LIN {X 0,Y 101.376,Z 372.445,A -85,B 0,C 180,E1 -29319.712,E2 -29319.712} C_VEL
LIN {X 0,Y 101.668,Z 372.001,A -85,B 0,C 180,E1 -29323.941,E2 -29323.941} C_VEL
LIN {X 0,Y 92.966,Z 374.596,A -85,B 0,C 180,E1 -29326.884,E2 -29326.884} C_VEL
LIN {X 0,Y 84.662,Z 376.417,A -85,B 0,C 180,E1 -29330.435,E2 -29330.435} C_VEL
LIN {X 0,Y 76.767,Z 377.474,A -85,B 0,C 180,E1 -29334.739,E2 -29334.739} C_VEL
LIN {X 0,Y 69.451,Z 377.857,A -85,B 0,C 180,E1 -29339.99,E2 -29339.99} C_VEL
LIN {X 0,Y 62.844,Z 377.562,A -85,B 0,C 180,E1 -29346.41,E2 -29346.41} C_VEL
LIN {X 0,Y 57.18,Z 376.524,A -85,B 0,C 180,E1 -29354.218,E2 -29354.218} C_VEL
LIN {X 0,Y 51.191,Z 373.837,A -85,B 0,C 180,E1 -29367.967,E2 -29367.967} C_VEL
LIN {X 0,Y 48.505,Z 369.652,A -85,B 0,C 180,E1 -29383.582,E2 -29383.582} C_VEL
LIN {X 0,Y 49.289,Z 364.241,A -85,B 0,C 180,E1 -29398.79,E2 -29398.79} C_VEL
LIN {X 0,Y 52.121,Z 358.398,A -85,B 0,C 180,E1 -29410.672,E2 -29410.672} C_VEL
LIN {X 0,Y 56.794,Z 350.599,A -85,B 0,C 180,E1 -29421.784,E2 -29421.784} C_VEL
LIN {X 0,Y 62.197,Z 342.135,A -85,B 0,C 180,E1 -29430.004,E2 -29430.004} C_VEL
LIN {X 0,Y 68.349,Z 332.145,A -85,B 0,C 180,E1 -29436.646,E2 -29436.646} C_VEL
LIN {X 0,Y 70.549,Z 328.315,A -85,B 0,C 180,E1 -29438.597,E2 -29438.597} C_VEL
LIN {X 0,Y 71.058,Z 326.204,A -85,B 0,C 180,E1 -29439.97,E2 -29439.97} C_VEL
LIN {X 0,Y 70.945,Z 321.655,A -85,B 0,C 180,E1 -29443.65,E2 -29443.65} C_VEL
LIN {X 0,Y 69.588,Z 315.642,A -85,B 0,C 180,E1 -29449.36,E2 -29449.36} C_VEL
LIN {X 0,Y 68.088,Z 310.944,A -85,B 0,C 180,E1 -29454.389,E2 -29454.389} C_VEL
LIN {X 0,Y 65.675,Z 304.781,A -85,B 0,C 180,E1 -29462.352,E2 -29462.352} C_VEL
LIN {X 0,Y 64.408,Z 302.022,A -85,B 0,C 180,E1 -29466.637,E2 -29466.637} C_VEL
LIN {X 0,Y 62.967,Z 299.24,A -85,B 0,C 180,E1 -29472.047,E2 -29472.047} C_VEL
LIN {X 0,Y 61.858,Z 297.335,A -85,B 0,C 180,E1 -29477.04,E2 -29477.04} C_VEL
LIN {X 0,Y 60.658,Z 294.989,A -85,B 0,C 180,E1 -29484.612,E2 -29484.612} C_VEL
LIN {X 0,Y 60.117,Z 293.628,A -85,B 0,C 180,E1 -29492.133,E2 -29492.133} C_VEL
LIN {X 0,Y 59.933,Z 293.549,A -85,B 0,C 180,E1 -29496.323,E2 -29496.323} C_VEL
LIN {X 0,Y 59.9,Z 293.87,A -85,B 0,C 180,E1 -29500.083,E2 -29500.083} C_VEL
LIN {X 0,Y 59.854,Z 295.517,A -85,B 0,C 180,E1 -29505.551,E2 -29505.551} C_VEL
LIN {X 0,Y 59.837,Z 298.087,A -85,B 0,C 180,E1 -29510.732,E2 -29510.732} C_VEL
LIN {X 0,Y 60.775,Z 306.566,A -85,B 0,C 180,E1 -29524.239,E2 -29524.239} C_VEL
LIN {X 0,Y 62.482,Z 311.333,A -85,B 0,C 180,E1 -29531.695,E2 -29531.695} C_VEL
LIN {X 0,Y 63.165,Z 317.36,A -85,B 0,C 180,E1 -29537.828,E2 -29537.828} C_VEL
LIN {X 0,Y 63.678,Z 323.437,A -85,B 0,C 180,E1 -29543.476,E2 -29543.476} C_VEL
LIN {X 0,Y 63.761,Z 326.496,A -85,B 0,C 180,E1 -29546.172,E2 -29546.172} C_VEL
LIN {X 0,Y 61.096,Z 335.145,A -85,B 0,C 180,E1 -29551.96,E2 -29551.96} C_VEL
LIN {X 0,Y 57.447,Z 345.258,A -85,B 0,C 180,E1 -29560.301,E2 -29560.301} C_VEL
LIN {X 0,Y 52.167,Z 353.065,A -85,B 0,C 180,E1 -29567.648,E2 -29567.648} C_VEL
LIN {X 0,Y 46.874,Z 360.782,A -85,B 0,C 180,E1 -29578.342,E2 -29578.342} C_VEL
LIN {X 0,Y 43.524,Z 366.979,A -85,B 0,C 180,E1 -29591.154,E2 -29591.154} C_VEL
LIN {X 0,Y 42.441,Z 371.361,A -85,B 0,C 180,E1 -29603.627,E2 -29603.627} C_VEL
LIN {X 0,Y 42.484,Z 373.184,A -85,B 0,C 180,E1 -29609.995,E2 -29609.995} C_VEL
LIN {X 0,Y 42.483,Z 375.384,A -85,B 0,C 180,E1 -29619.517,E2 -29619.517} C_VEL
LIN {X 0,Y 45.164,Z 378.472,A -85,B 0,C 180,E1 -29637.823,E2 -29637.823} C_VEL
LIN {X 0,Y 51.747,Z 380.173,A -85,B 0,C 180,E1 -29652.765,E2 -29652.765} C_VEL
LIN {X 0,Y 61.206,Z 380.584,A -85,B 0,C 180,E1 -29663.486,E2 -29663.486} C_VEL
LIN {X 0,Y 72.265,Z 379.685,A -85,B 0,C 180,E1 -29671.072,E2 -29671.072} C_VEL
LIN {X 0,Y 84.324,Z 377.434,A -85,B 0,C 180,E1 -29676.455,E2 -29676.455} C_VEL
LIN {X 0,Y 93.014,Z 375.129,A -85,B 0,C 180,E1 -29679.177,E2 -29679.177} C_VEL
LIN {X 0,Y 94.648,Z 374.479,A -85,B 0,C 180,E1 -29681.102,E2 -29681.102} C_VEL
LIN {X 0,Y 92.095,Z 375.088,A -85,B 0,C 180,E1 -29682.219,E2 -29682.219} C_VEL
LIN {X 0,Y 79.337,Z 377.481,A -85,B 0,C 180,E1 -29687.001,E2 -29687.001} C_VEL
LIN {X 0,Y 66.834,Z 378.352,A -85,B 0,C 180,E1 -29693.954,E2 -29693.954} C_VEL
LIN {X 0,Y 56.312,Z 377.664,A -85,B 0,C 180,E1 -29703.283,E2 -29703.283} C_VEL
LIN {X 0,Y 47.446,Z 375.304,A -85,B 0,C 180,E1 -29717.218,E2 -29717.218} C_VEL
LIN {X 0,Y 42.406,Z 371.584,A -85,B 0,C 180,E1 -29734.048,E2 -29734.048} C_VEL
LIN {X 0,Y 41.468,Z 366.499,A -85,B 0,C 180,E1 -29752.482,E2 -29752.482} C_VEL
LIN {X 0,Y 44.089,Z 360.223,A -85,B 0,C 180,E1 -29768.761,E2 -29768.761} C_VEL
LIN {X 0,Y 48.727,Z 352.886,A -85,B 0,C 180,E1 -29781.712,E2 -29781.712} C_VEL
LIN {X 0,Y 54.251,Z 344.899,A -85,B 0,C 180,E1 -29791.12,E2 -29791.12} C_VEL
LIN {X 0,Y 60.441,Z 335.662,A -85,B 0,C 180,E1 -29798.363,E2 -29798.363} C_VEL
LIN {X 0,Y 64.978,Z 328.329,A -85,B 0,C 180,E1 -29802.496,E2 -29802.496} C_VEL
LIN {X 0,Y 65.059,Z 324.8,A -85,B 0,C 180,E1 -29805.668,E2 -29805.668} C_VEL
LIN {X 0,Y 63.918,Z 318.451,A -85,B 0,C 180,E1 -29812.522,E2 -29812.522} C_VEL
LIN {X 0,Y 62.176,Z 312.612,A -85,B 0,C 180,E1 -29820.229,E2 -29820.229} C_VEL
LIN {X 0,Y 60.848,Z 308.888,A -85,B 0,C 180,E1 -29826.07,E2 -29826.07} C_VEL
LIN {X 0,Y 59.187,Z 304.804,A -85,B 0,C 180,E1 -29834.582,E2 -29834.582} C_VEL
LIN {X 0,Y 57.933,Z 302.351,A -85,B 0,C 180,E1 -29842.674,E2 -29842.674} C_VEL
LIN {X 0,Y 57.449,Z 300.523,A -85,B 0,C 180,E1 -29850.717,E2 -29850.717} C_VEL
LIN {X 0,Y 57.346,Z 300.105,A -85,B 0,C 180,E1 -29858.441,E2 -29858.441} C_VEL
LIN {X 0,Y 57.988,Z 300.172,A -85,B 0,C 180,E1 -29865.984,E2 -29865.984} C_VEL
LIN {X 0,Y 59.389,Z 302.981,A -85,B 0,C 180,E1 -29876.77,E2 -29876.77} C_VEL
LIN {X 0,Y 60.008,Z 304.274,A -85,B 0,C 180,E1 -29880.011,E2 -29880.011} C_VEL
LIN {X 0,Y 60.775,Z 306.566,A -85,B 0,C 180,E1 -29884.239,E2 -29884.239} C_VEL
LIN {X 0,Y 61.035,Z 308.99,A -85,B 0,C 180,E1 -29887.101,E2 -29887.101} C_VEL
LIN {X 0,Y 60.582,Z 312.079,A -85,B 0,C 180,E1 -29889.423,E2 -29889.423} C_VEL
LIN {X 0,Y 58.208,Z 321.047,A -85,B 0,C 180,E1 -29895.157,E2 -29895.157} C_VEL
LIN {X 0,Y 58.018,Z 323.039,A -85,B 0,C 180,E1 -29897.019,E2 -29897.019} C_VEL
LIN {X 0,Y 57.98,Z 328.126,A -85,B 0,C 180,E1 -29902.271,E2 -29902.271} C_VEL
LIN {X 0,Y 57.244,Z 330.798,A -85,B 0,C 180,E1 -29904.321,E2 -29904.321} C_VEL
LIN {X 0,Y 52.946,Z 341.495,A -85,B 0,C 180,E1 -29912.829,E2 -29912.829} C_VEL
LIN {X 0,Y 50.774,Z 346.122,A -85,B 0,C 180,E1 -29917.252,E2 -29917.252} C_VEL
LIN {X 0,Y 44.967,Z 353.729,A -85,B 0,C 180,E1 -29925.3,E2 -29925.3} C_VEL
LIN {X 0,Y 39.392,Z 361.175,A -85,B 0,C 180,E1 -29937.633,E2 -29937.633} C_VEL
LIN {X 0,Y 36.106,Z 367.154,A -85,B 0,C 180,E1 -29953.018,E2 -29953.018} C_VEL
LIN {X 0,Y 35.457,Z 371.851,A -85,B 0,C 180,E1 -29969.994,E2 -29969.994} C_VEL
LIN {X 0,Y 35.593,Z 374.171,A -85,B 0,C 180,E1 -29981.382,E2 -29981.382} C_VEL
LIN {X 0,Y 39.045,Z 377.526,A -85,B 0,C 180,E1 -30002.676,E2 -30002.676} C_VEL
LIN {X 0,Y 46.782,Z 379.462,A -85,B 0,C 180,E1 -30018.682,E2 -30018.682} C_VEL
LIN {X 0,Y 57.258,Z 380.093,A -85,B 0,C 180,E1 -30029.219,E2 -30029.219} C_VEL
LIN {X 0,Y 69.1,Z 379.434,A -85,B 0,C 180,E1 -30036.25,E2 -30036.25} C_VEL
LIN {X 0,Y 76.896,Z 378.399,A -85,B 0,C 180,E1 -30039.399,E2 -30039.399} C_VEL
LIN {X 0,Y 79.384,Z 377.862,A -85,B 0,C 180,E1 -30041.184,E2 -30041.184} C_VEL
LIN {X 0,Y 73.286,Z 378.502,A -85,B 0,C 180,E1 -30043.52,E2 -30043.52} C_VEL
LIN {X 0,Y 64.738,Z 378.844,A -85,B 0,C 180,E1 -30047.682,E2 -30047.682} C_VEL
LIN {X 0,Y 56.628,Z 378.527,A -85,B 0,C 180,E1 -30053.12,E2 -30053.12} C_VEL
LIN {X 0,Y 49.192,Z 377.474,A -85,B 0,C 180,E1 -30060.285,E2 -30060.285} C_VEL
LIN {X 0,Y 40.091,Z 374.649,A -85,B 0,C 180,E1 -30075.411,E2 -30075.411} C_VEL
LIN {X 0,Y 34.869,Z 370.186,A -85,B 0,C 180,E1 -30096.283,E2 -30096.283} C_VEL
LIN {X 0,Y 34.506,Z 365.614,A -85,B 0,C 180,E1 -30114.522,E2 -30114.522} C_VEL
LIN {X 0,Y 37.141,Z 360.075,A -85,B 0,C 180,E1 -30131.049,E2 -30131.049} C_VEL
LIN {X 0,Y 42.284,Z 352.781,A -85,B 0,C 180,E1 -30145.527,E2 -30145.527} C_VEL
LIN {X 0,Y 48.562,Z 344.479,A -85,B 0,C 180,E1 -30155.796,E2 -30155.796} C_VEL
LIN {X 0,Y 55.826,Z 334.353,A -85,B 0,C 180,E1 -30163.657,E2 -30163.657} C_VEL
LIN {X 0,Y 58.412,Z 330.512,A -85,B 0,C 180,E1 -30165.778,E2 -30165.778} C_VEL
LIN {X 0,Y 59.119,Z 329.025,A -85,B 0,C 180,E1 -30166.804,E2 -30166.804} C_VEL
LIN {X 0,Y 58.927,Z 325.419,A -85,B 0,C 180,E1 -30170.969,E2 -30170.969} C_VEL
LIN {X 0,Y 58.196,Z 320.601,A -85,B 0,C 180,E1 -30177.339,E2 -30177.339} C_VEL
LIN {X 0,Y 56.756,Z 314.985,A -85,B 0,C 180,E1 -30186.416,E2 -30186.416} C_VEL
LIN {X 0,Y 56.051,Z 312.648,A -85,B 0,C 180,E1 -30191.227,E2 -30191.227} C_VEL
LIN {X 0,Y 55.463,Z 310.664,A -85,B 0,C 180,E1 -30196.085,E2 -30196.085} C_VEL
LIN {X 0,Y 54.67,Z 308.732,A -85,B 0,C 180,E1 -30202.851,E2 -30202.851} C_VEL
LIN {X 0,Y 54.427,Z 307.364,A -85,B 0,C 180,E1 -30208.916,E2 -30208.916} C_VEL
LIN {X 0,Y 54.338,Z 306.635,A -85,B 0,C 180,E1 -30217.183,E2 -30217.183} C_VEL
LIN {X 0,Y 54.913,Z 306.605,A -85,B 0,C 180,E1 -30225.182,E2 -30225.182} C_VEL
LIN {X 0,Y 55.597,Z 308.283,A -85,B 0,C 180,E1 -30232.75,E2 -30232.75} C_VEL
LIN {X 0,Y 56.265,Z 309.927,A -85,B 0,C 180,E1 -30237.916,E2 -30237.916} C_VEL
LIN {X 0,Y 57.517,Z 314.761,A -85,B 0,C 180,E1 -30247.03,E2 -30247.03} C_VEL
LIN {X 0,Y 57.896,Z 317.176,A -85,B 0,C 180,E1 -30250.503,E2 -30250.503} C_VEL
LIN {X 0,Y 58.018,Z 323.039,A -85,B 0,C 180,E1 -30257.019,E2 -30257.019} C_VEL
LIN {X 0,Y 57.549,Z 325.508,A -85,B 0,C 180,E1 -30259.023,E2 -30259.023} C_VEL
LIN {X 0,Y 55.656,Z 329.233,A -85,B 0,C 180,E1 -30260.903,E2 -30260.903} C_VEL
LIN {X 0,Y 49.305,Z 337.8,A -85,B 0,C 180,E1 -30264.582,E2 -30264.582} C_VEL
LIN {X 0,Y 48.081,Z 339.855,A -85,B 0,C 180,E1 -30266.242,E2 -30266.242} C_VEL
LIN {X 0,Y 45.401,Z 345.135,A -85,B 0,C 180,E1 -30271.627,E2 -30271.627} C_VEL
LIN {X 0,Y 39.053,Z 352.866,A -85,B 0,C 180,E1 -30280.1,E2 -30280.1} C_VEL
LIN {X 0,Y 32.747,Z 360.402,A -85,B 0,C 180,E1 -30293.822,E2 -30293.822} C_VEL
LIN {X 0,Y 29.444,Z 365.524,A -85,B 0,C 180,E1 -30309.012,E2 -30309.012} C_VEL
LIN {X 0,Y 28.429,Z 370.475,A -85,B 0,C 180,E1 -30329.992,E2 -30329.992} C_VEL
LIN {X 0,Y 28.76,Z 372.945,A -85,B 0,C 180,E1 -30344.137,E2 -30344.137} C_VEL
LIN {X 0,Y 33.311,Z 376.481,A -85,B 0,C 180,E1 -30369.259,E2 -30369.259} C_VEL
LIN {X 0,Y 42.435,Z 378.664,A -85,B 0,C 180,E1 -30385.893,E2 -30385.893} C_VEL
LIN {X 0,Y 53.965,Z 379.572,A -85,B 0,C 180,E1 -30395.722,E2 -30395.722} C_VEL
LIN {X 0,Y 62.944,Z 379.398,A -85,B 0,C 180,E1 -30400.419,E2 -30400.419} C_VEL
LIN {X 0,Y 58.675,Z 379.227,A -85,B 0,C 180,E1 -30403.365,E2 -30403.365} C_VEL
LIN {X 0,Y 46.993,Z 378.008,A -85,B 0,C 180,E1 -30411.384,E2 -30411.384} C_VEL
LIN {X 0,Y 39.384,Z 376.302,A -85,B 0,C 180,E1 -30419.983,E2 -30419.983} C_VEL
LIN {X 0,Y 32.992,Z 373.86,A -85,B 0,C 180,E1 -30432.278,E2 -30432.278} C_VEL
LIN {X 0,Y 28.488,Z 370.519,A -85,B 0,C 180,E1 -30449.537,E2 -30449.537} C_VEL
LIN {X 0,Y 27.448,Z 365.231,A -85,B 0,C 180,E1 -30475.255,E2 -30475.255} C_VEL
LIN {X 0,Y 30.926,Z 358.96,A -85,B 0,C 180,E1 -30496.872,E2 -30496.872} C_VEL
LIN {X 0,Y 37.178,Z 351.26,A -85,B 0,C 180,E1 -30512.715,E2 -30512.715} C_VEL
LIN {X 0,Y 43.942,Z 343.174,A -85,B 0,C 180,E1 -30522.467,E2 -30522.467} C_VEL
LIN {X 0,Y 51.682,Z 333.139,A -85,B 0,C 180,E1 -30529.725,E2 -30529.725} C_VEL
LIN {X 0,Y 53.358,Z 330.526,A -85,B 0,C 180,E1 -30531.279,E2 -30531.279} C_VEL
LIN {X 0,Y 53.05,Z 325.542,A -85,B 0,C 180,E1 -30538.53,E2 -30538.53} C_VEL
LIN {X 0,Y 52.393,Z 321.069,A -85,B 0,C 180,E1 -30546.427,E2 -30546.427} C_VEL
LIN {X 0,Y 51.857,Z 318.242,A -85,B 0,C 180,E1 -30552.665,E2 -30552.665} C_VEL
LIN {X 0,Y 51.245,Z 315.541,A -85,B 0,C 180,E1 -30560.607,E2 -30560.607} C_VEL
LIN {X 0,Y 50.945,Z 314.221,A -85,B 0,C 180,E1 -30566.525,E2 -30566.525} C_VEL
LIN {X 0,Y 51.021,Z 312.978,A -85,B 0,C 180,E1 -30575.606,E2 -30575.606} C_VEL
LIN {X 0,Y 51.492,Z 312.9,A -85,B 0,C 180,E1 -30584.172,E2 -30584.172} C_VEL
LIN {X 0,Y 52.028,Z 314.51,A -85,B 0,C 180,E1 -30592.25,E2 -30592.25} C_VEL
LIN {X 0,Y 52.444,Z 316.341,A -85,B 0,C 180,E1 -30597.764,E2 -30597.764} C_VEL
LIN {X 0,Y 53.061,Z 320.142,A -85,B 0,C 180,E1 -30605.48,E2 -30605.48} C_VEL
LIN {X 0,Y 52.849,Z 324.932,A -85,B 0,C 180,E1 -30611.743,E2 -30611.743} C_VEL
LIN {X 0,Y 52.451,Z 329.743,A -85,B 0,C 180,E1 -30617.56,E2 -30617.56} C_VEL
LIN {X 0,Y 51.736,Z 332.141,A -85,B 0,C 180,E1 -30619.799,E2 -30619.799} C_VEL
LIN {X 0,Y 48.081,Z 339.855,A -85,B 0,C 180,E1 -30626.242,E2 -30626.242} C_VEL
LIN {X 0,Y 46.449,Z 342.251,A -85,B 0,C 180,E1 -30628.08,E2 -30628.08} C_VEL
LIN {X 0,Y 43.135,Z 345.262,A -85,B 0,C 180,E1 -30629.604,E2 -30629.604} C_VEL
LIN {X 0,Y 35.349,Z 350.71,A -85,B 0,C 180,E1 -30632.006,E2 -30632.006} C_VEL
LIN {X 0,Y 32.497,Z 353.138,A -85,B 0,C 180,E1 -30634.747,E2 -30634.747} C_VEL
LIN {X 0,Y 25.389,Z 360.695,A -85,B 0,C 180,E1 -30651.465,E2 -30651.465} C_VEL
LIN {X 0,Y 21.546,Z 366.973,A -85,B 0,C 180,E1 -30678.258,E2 -30678.258} C_VEL
LIN {X 0,Y 21.441,Z 368.975,A -85,B 0,C 180,E1 -30689.99,E2 -30689.99} C_VEL
LIN {X 0,Y 22.05,Z 371.577,A -85,B 0,C 180,E1 -30708.575,E2 -30708.575} C_VEL
LIN {X 0,Y 28.194,Z 375.421,A -85,B 0,C 180,E1 -30738.389,E2 -30738.389} C_VEL
LIN {X 0,Y 38.907,Z 377.825,A -85,B 0,C 180,E1 -30754.566,E2 -30754.566} C_VEL
LIN {X 0,Y 45.062,Z 378.554,A -85,B 0,C 180,E1 -30759.341,E2 -30759.341} C_VEL
LIN {X 0,Y 45.69,Z 378.479,A -85,B 0,C 180,E1 -30762.068,E2 -30762.068} C_VEL
LIN {X 0,Y 35.607,Z 376.387,A -85,B 0,C 180,E1 -30770.674,E2 -30770.674} C_VEL
LIN {X 0,Y 28.132,Z 373.851,A -85,B 0,C 180,E1 -30782.357,E2 -30782.357} C_VEL
LIN {X 0,Y 20.786,Z 368.684,A -85,B 0,C 180,E1 -30812.335,E2 -30812.335} C_VEL
LIN {X 0,Y 21.118,Z 363.041,A -85,B 0,C 180,E1 -30845.43,E2 -30845.43} C_VEL
LIN {X 0,Y 25.487,Z 357.468,A -85,B 0,C 180,E1 -30866.239,E2 -30866.239} C_VEL
LIN {X 0,Y 33.01,Z 349.454,A -85,B 0,C 180,E1 -30882.299,E2 -30882.299} C_VEL
LIN {X 0,Y 40.959,Z 340.654,A -85,B 0,C 180,E1 -30891.391,E2 -30891.391} C_VEL
LIN {X 0,Y 47.521,Z 332.553,A -85,B 0,C 180,E1 -30896.344,E2 -30896.344} C_VEL
LIN {X 0,Y 47.721,Z 329.272,A -85,B 0,C 180,E1 -30901.832,E2 -30901.832} C_VEL
LIN {X 0,Y 47.487,Z 324.406,A -85,B 0,C 180,E1 -30912.291,E2 -30912.291} C_VEL
LIN {X 0,Y 47.305,Z 322.408,A -85,B 0,C 180,E1 -30917.981,E2 -30917.981} C_VEL
LIN {X 0,Y 47.172,Z 320.959,A -85,B 0,C 180,E1 -30923.438,E2 -30923.438} C_VEL
LIN {X 0,Y 47.194,Z 319.414,A -85,B 0,C 180,E1 -30933.481,E2 -30933.481} C_VEL
LIN {X 0,Y 47.714,Z 318.988,A -85,B 0,C 180,E1 -30942.882,E2 -30942.882} C_VEL
LIN {X 0,Y 48.081,Z 320.556,A -85,B 0,C 180,E1 -30951.609,E2 -30951.609} C_VEL
LIN {X 0,Y 48.238,Z 321.858,A -85,B 0,C 180,E1 -30955.837,E2 -30955.837} C_VEL
LIN {X 0,Y 48.352,Z 324.569,A -85,B 0,C 180,E1 -30962.096,E2 -30962.096} C_VEL
LIN {X 0,Y 47.654,Z 328.935,A -85,B 0,C 180,E1 -30968.495,E2 -30968.495} C_VEL
LIN {X 0,Y 46.864,Z 332.984,A -85,B 0,C 180,E1 -30973.882,E2 -30973.882} C_VEL
LIN {X 0,Y 41.751,Z 342.109,A -85,B 0,C 180,E1 -30982.194,E2 -30982.194} C_VEL
LIN {X 0,Y 39.199,Z 345.939,A -85,B 0,C 180,E1 -30986.293,E2 -30986.293} C_VEL
LIN {X 0,Y 32.497,Z 353.138,A -85,B 0,C 180,E1 -30994.747,E2 -30994.747} C_VEL
LIN {X 0,Y 28.733,Z 356.603,A -85,B 0,C 180,E1 -31000.251,E2 -31000.251} C_VEL
LIN {X 0,Y 24.534,Z 359.642,A -85,B 0,C 180,E1 -31006.464,E2 -31006.464} C_VEL
LIN {X 0,Y 16.629,Z 364.768,A -85,B 0,C 180,E1 -31027.546,E2 -31027.546} C_VEL
LIN {X 0,Y 14.435,Z 367.83,A -85,B 0,C 180,E1 -31053.837,E2 -31053.837} C_VEL
LIN {X 0,Y 15.594,Z 370.192,A -85,B 0,C 180,E1 -31076.771,E2 -31076.771} C_VEL
LIN {X 0,Y 24.106,Z 374.231,A -85,B 0,C 180,E1 -31110.984,E2 -31110.984} C_VEL
LIN {X 0,Y 30.043,Z 375.729,A -85,B 0,C 180,E1 -31119.326,E2 -31119.326} C_VEL
LIN {X 0,Y 29.45,Z 375.451,A -85,B 0,C 180,E1 -31122.636,E2 -31122.636} C_VEL
LIN {X 0,Y 19.096,Z 371.54,A -85,B 0,C 180,E1 -31139.965,E2 -31139.965} C_VEL
LIN {X 0,Y 13.065,Z 365.87,A -85,B 0,C 180,E1 -31184.538,E2 -31184.538} C_VEL
LIN {X 0,Y 15.973,Z 360.551,A -85,B 0,C 180,E1 -31222.867,E2 -31222.867} C_VEL
LIN {X 0,Y 22.889,Z 354.109,A -85,B 0,C 180,E1 -31244.108,E2 -31244.108} C_VEL
LIN {X 0,Y 32.039,Z 345.503,A -85,B 0,C 180,E1 -31256.029,E2 -31256.029} C_VEL
LIN {X 0,Y 41.107,Z 335.634,A -85,B 0,C 180,E1 -31262.581,E2 -31262.581} C_VEL
LIN {X 0,Y 41.896,Z 334.711,A -85,B 0,C 180,E1 -31263.023,E2 -31263.023} C_VEL
LIN {X 0,Y 42.355,Z 333.845,A -85,B 0,C 180,E1 -31263.968,E2 -31263.968} C_VEL
LIN {X 0,Y 42.632,Z 330.715,A -85,B 0,C 180,E1 -31271.262,E2 -31271.262} C_VEL
LIN {X 0,Y 42.84,Z 327.994,A -85,B 0,C 180,E1 -31279.01,E2 -31279.01} C_VEL
LIN {X 0,Y 42.954,Z 326.59,A -85,B 0,C 180,E1 -31284.901,E2 -31284.901} C_VEL
LIN {X 0,Y 42.986,Z 325.807,A -85,B 0,C 180,E1 -31290.646,E2 -31290.646} C_VEL
LIN {X 0,Y 43.547,Z 324.982,A -85,B 0,C 180,E1 -31301.186,E2 -31301.186} C_VEL
LIN {X 0,Y 43.665,Z 325.306,A -85,B 0,C 180,E1 -31304.971,E2 -31304.971} C_VEL
LIN {X 0,Y 43.836,Z 326.343,A -85,B 0,C 180,E1 -31310.79,E2 -31310.79} C_VEL
LIN {X 0,Y 43.657,Z 328.736,A -85,B 0,C 180,E1 -31317.709,E2 -31317.709} C_VEL
LIN {X 0,Y 42.85,Z 331.543,A -85,B 0,C 180,E1 -31322.589,E2 -31322.589} C_VEL
LIN {X 0,Y 41.904,Z 334.612,A -85,B 0,C 180,E1 -31327.413,E2 -31327.413} C_VEL
LIN {X 0,Y 36.438,Z 342.908,A -85,B 0,C 180,E1 -31335.32,E2 -31335.32} C_VEL
LIN {X 0,Y 34.993,Z 344.851,A -85,B 0,C 180,E1 -31337.426,E2 -31337.426} C_VEL
LIN {X 0,Y 27.28,Z 352.44,A -85,B 0,C 180,E1 -31345.599,E2 -31345.599} C_VEL
LIN {X 0,Y 19.174,Z 359.825,A -85,B 0,C 180,E1 -31362.837,E2 -31362.837} C_VEL
LIN {X 0,Y 14.43,Z 366.386,A -85,B 0,C 180,E1 -31401.308,E2 -31401.308} C_VEL
LIN {X 0,Y 14.435,Z 367.83,A -85,B 0,C 180,E1 -31413.837,E2 -31413.837} C_VEL
LIN {X 0,Y 13.861,Z 368.289,A -85,B 0,C 180,E1 -31420.094,E2 -31420.094} C_VEL
LIN {X 0,Y 11.718,Z 368.327,A -85,B 0,C 180,E1 -31429.427,E2 -31429.427} C_VEL
LIN {X 0,Y 9.217,Z 367.862,A -85,B 0,C 180,E1 -31438.174,E2 -31438.174} C_VEL
LIN {X 0,Y 5.465,Z 366.678,A -85,B 0,C 180,E1 -31457.17,E2 -31457.17} C_VEL
LIN {X 0,Y 3.851,Z 363.643,A -85,B 0,C 180,E1 -31568.822,E2 -31568.822} C_VEL
LIN {X 0,Y 9.513,Z 360.341,A -85,B 0,C 180,E1 -31601.74,E2 -31601.74} C_VEL
LIN {X 0,Y 13.313,Z 357.773,A -85,B 0,C 180,E1 -31611.05,E2 -31611.05} C_VEL
LIN {X 0,Y 22.257,Z 350.811,A -85,B 0,C 180,E1 -31623.557,E2 -31623.557} C_VEL
LIN {X 0,Y 31.813,Z 342.097,A -85,B 0,C 180,E1 -31629.439,E2 -31629.439} C_VEL
LIN {X 0,Y 37.122,Z 336.519,A -85,B 0,C 180,E1 -31631.508,E2 -31631.508} C_VEL
LIN {X 0,Y 37.612,Z 335.258,A -85,B 0,C 180,E1 -31634.492,E2 -31634.492} C_VEL
LIN {X 0,Y 38.229,Z 332.848,A -85,B 0,C 180,E1 -31642.566,E2 -31642.566} C_VEL
LIN {X 0,Y 38.501,Z 331.963,A -85,B 0,C 180,E1 -31646.818,E2 -31646.818} C_VEL
LIN {X 0,Y 38.987,Z 330.906,A -85,B 0,C 180,E1 -31658.886,E2 -31658.886} C_VEL
LIN {X 0,Y 39.238,Z 331.97,A -85,B 0,C 180,E1 -31669.7,E2 -31669.7} C_VEL
LIN {X 0,Y 38.66,Z 333.816,A -85,B 0,C 180,E1 -31674.803,E2 -31674.803} C_VEL
LIN {X 0,Y 37.17,Z 336.885,A -85,B 0,C 180,E1 -31680.018,E2 -31680.018} C_VEL
LIN {X 0,Y 31.818,Z 343.659,A -85,B 0,C 180,E1 -31686.233,E2 -31686.233} C_VEL
LIN {X 0,Y 28.443,Z 347.028,A -85,B 0,C 180,E1 -31688.707,E2 -31688.707} C_VEL
LIN {X 0,Y 18.442,Z 355.392,A -85,B 0,C 180,E1 -31697.654,E2 -31697.654} C_VEL
LIN {X 0,Y 9.761,Z 362.102,A -85,B 0,C 180,E1 -31723.913,E2 -31723.913} C_VEL
LIN {X 0,Y 7.537,Z 366.381,A -85,B 0,C 180,E1 -31780.834,E2 -31780.834} C_VEL
LIN {X 0,Y 9.898,Z 368.675,A -85,B 0,C 180,E1 -31815.208,E2 -31815.208} C_VEL
LIN {X 0,Y 15.217,Z 371.04,A -85,B 0,C 180,E1 -31837.433,E2 -31837.433} C_VEL
LIN {X 0,Y 14.911,Z 370.863,A -85,B 0,C 180,E1 -31840.458,E2 -31840.458} C_VEL
LIN {X 0,Y 6.024,Z 364.608,A -85,B 0,C 180,E1 -31909.155,E2 -31909.155} C_VEL
LIN {X 0,Y 13.313,Z 357.773,A -85,B 0,C 180,E1 -31971.05,E2 -31971.05} C_VEL
LIN {X 0,Y 15.945,Z 355.538,A -85,B 0,C 180,E1 -31978.645,E2 -31978.645} C_VEL
LIN {X 0,Y 19.715,Z 351.64,A -85,B 0,C 180,E1 -31991.48,E2 -31991.48} C_VEL
LIN {X 0,Y 23.921,Z 347.478,A -85,B 0,C 180,E1 -32000.262,E2 -32000.262} C_VEL
LIN {X 0,Y 26.809,Z 344.745,A -85,B 0,C 180,E1 -32002.025,E2 -32002.025} C_VEL
LIN {X 0,Y 32.197,Z 339.518,A -85,B 0,C 180,E1 -32002.316,E2 -32002.316} C_VEL
LIN {X 0,Y 33.119,Z 338.486,A -85,B 0,C 180,E1 -32002.738,E2 -32002.738} C_VEL
LIN {X 0,Y 33.587,Z 337.566,A -85,B 0,C 180,E1 -32006.835,E2 -32006.835} C_VEL
LIN {X 0,Y 34.136,Z 336.589,A -85,B 0,C 180,E1 -32015.706,E2 -32015.706} C_VEL
LIN {X 0,Y 34.143,Z 337.493,A -85,B 0,C 180,E1 -32028.142,E2 -32028.142} C_VEL
LIN {X 0,Y 33.426,Z 338.574,A -85,B 0,C 180,E1 -32030.265,E2 -32030.265} C_VEL
LIN {X 0,Y 28.258,Z 344.293,A -85,B 0,C 180,E1 -32034.241,E2 -32034.241} C_VEL
LIN {X 0,Y 19.397,Z 351.766,A -85,B 0,C 180,E1 -32035.255,E2 -32035.255} C_VEL
LIN {X 0,Y 9.736,Z 358.483,A -85,B 0,C 180,E1 -32037.211,E2 -32037.211} C_VEL
LIN {X 0,Y 4.626,Z 361.522,A -85,B 0,C 180,E1 -32040.146,E2 -32040.146} C_VEL
LIN {X 0,Y 1.5,Z 363.128,A -85,B 0,C 180,E1 -32040.449,E2 -32040.449} C_VEL
LIN {X 0,Y 13.363,Z 355.552,A -85,B 0,C 180,E1 -32002.429,E2 -32002.429} C_VEL
LIN {X 0,Y 22.777,Z 348.313,A -85,B 0,C 180,E1 -32001.933,E2 -32001.933} C_VEL
LIN {X 0,Y 26.809,Z 344.745,A -85,B 0,C 180,E1 -32002.025,E2 -32002.025} C_VEL
LIN {X 0,Y 30.153,Z 346.226,A -85,B 0,C 180,E1 -32002.206,E2 -32002.206} C_VEL
LIN {X 0,Y 30.153,Z 600,A -85,B 0,C 180,E1 -32002.206,E2 -32002.206} C_VEL
LIN {X 0,Y 30.153,Z 600,A -85,B 0,C 180,E1 -32002.206,E2 -32002.206}

QRS_NEXT_CUT()

QRS_NEXT()
QRS_HOME()

END
